# B&R Automation Studio project Sortering_af_Kasser_med_robot1
Automation Studio 4.7.2.98

## Configuration Config1

### Hardware
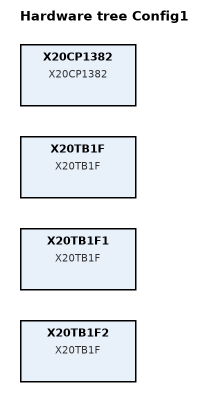
```
X20CP1382 : X20CP1382 v1.8.0.0  [X1 -> X1.SL; X2 -> X2.SL; X3 -> X3.SL]
  Module X1 (Type=X1, Virtual=true, Version=1.8.0.0)
    Connection (Connector=SS1, TargetModule=X20TB1F, TargetConnector=SS)
    Connection (Connector=SL, TargetModule=X20CP1382, TargetConnector=X1)
  Module X2 (Type=X2, Virtual=true, Version=1.8.0.0)
    Connection (Connector=SS1, TargetModule=X20TB1F1, TargetConnector=SS)
    Connection (Connector=SL, TargetModule=X20CP1382, TargetConnector=X2)
  Module X3 (Type=X3, Virtual=true, Version=1.8.0.0)
    Connection (Connector=SS1, TargetModule=X20TB1F2, TargetConnector=SS)
    Connection (Connector=SL, TargetModule=X20CP1382, TargetConnector=X3)
  Connector IF2:
    ActivateDevice = 1
  ConfigurationID = Sortering_af_Kasser_med_robot_Config1
  Simulation = 1
X20TB1F : X20TB1F v1.0.0.0
X20TB1F1 : X20TB1F v1.0.0.0
X20TB1F2 : X20TB1F v1.0.0.0
```

## Logical view

### Program Logical/Controller (IEC)

#### Variables.var
```iecst
(*Input Variables*)
VAR
	diEaterSmall : BOOL;
	diEaterMedium : BOOL;
	diEaterLarge : BOOL;
	diWeight_activated : BOOL;
	diWeight_measurement : WORD;
END_VAR
(*Output Variables*)
VAR
	doRobotMoveRight : BOOL;
	doRobotActivate : BOOL;
	doBeltMotor1 : BOOL;
	doBeltMotor2 : BOOL;
	doBeltMotor3 : BOOL;
	doEaterSmall : WORD;
	doEaterMedium : WORD;
	doEaterLarge : WORD;
	doLightSmall : BOOL;
	doLightMedium : BOOL;
	doLightLarge : BOOL;
END_VAR
(*Function Blocks*)
VAR
	R_TRIG_Weight : R_TRIG;
	F_TRIG_Weight : F_TRIG;
	TON_Weight : TON;
	CTU_Small : CTU;
	CTU_Medium : CTU;
	CTU_Large : CTU;
END_VAR
```

#### Main.st
```iecst
PROGRAM _INIT
	doBeltMotor1 := TRUE;
	doBeltMotor2 := TRUE;
	doBeltMotor3 := TRUE;
	TON_Weight.PT := T#0.5s;

END_PROGRAM

PROGRAM _CYCLIC
	R_TRIG_Weight.CLK := diWeight_activated;
	F_TRIG_Weight.CLK := diWeight_activated;
	CTU_Small.CU := diEaterSmall;
	CTU_Medium.CU := diEaterMedium;
	CTU_Large.CU := diEaterLarge;

	// Box has entered the weight.
	IF R_TRIG_Weight.Q THEN
		// Default is we set timer to stop belt.
		TON_Weight.IN := TRUE;

		// Depending on bagage size, telling robot what to do.
		doRobotActivate := TRUE;
		IF diWeight_measurement < 5000 THEN
			doRobotMoveRight := TRUE;
		ELSIF diWeight_measurement < 7500 THEN
			doRobotMoveRight := FALSE;
		ELSE
			// Box can pass and Robot should do nothing.
			TON_Weight.IN := FALSE;
			doRobotActivate := FALSE;
		END_IF;

		// Setting correct light indicator
		IF diWeight_measurement < 5000 THEN
			doLightSmall := TRUE;
		ELSIF diWeight_measurement < 7500 THEN
			doLightMedium := TRUE;
		ELSE
			doLightLarge := TRUE;
		END_IF;
	END_IF;

	// Timer for box placement is done.
	IF TON_Weight.Q THEN
		// Box is in place to be picked up, stopping BeltMotor.
		doBeltMotor1 := FALSE;
		TON_Weight.IN := FALSE;
	END_IF;

	// Reset stuff.
	IF F_TRIG_Weight.Q THEN
		// Resetting lights.
		doLightSmall := FALSE;
		doLightMedium := FALSE;
		doLightLarge := FALSE;

		// Starting BeltMotor wether it's going or not.
		doBeltMotor1 := TRUE;

		// Setting Robot Activation to low
		doRobotActivate := FALSE;
	END_IF;

	// Update Counters.
	doEaterSmall := UINT_TO_WORD( CTU_Small.CV );
	doEaterMedium := UINT_TO_WORD( CTU_Medium.CV );
	doEaterLarge := UINT_TO_WORD( CTU_Large.CV );

	// Call Function Blocks.
	CTU_Small();
	CTU_Medium();
	CTU_Large();
	TON_Weight();
	R_TRIG_Weight();
	F_TRIG_Weight();
END_PROGRAM

PROGRAM _EXIT
	(* Insert code here *)

END_PROGRAM
```

Listed in the project but not available here: Logical/Global.typ, Logical/Global.var, Logical/Libraries
